INTERFACE I_MirrorCovers

METHOD Close : BOOL
VAR_INPUT
END_VAR
END_METHOD

PROPERTY Closed : BOOL
GET
END_GET
END_PROPERTY

PROPERTY Error : BOOL
GET
END_GET
END_PROPERTY

METHOD Open : BOOL
VAR_INPUT
END_VAR
END_METHOD

PROPERTY Opened : BOOL
GET
END_GET
END_PROPERTY

METHOD Reset : BOOL
VAR_INPUT
END_VAR
END_METHOD

END_INTERFACE

(* stored: Version 1.1.0.1, ProductVersion 3.1.4024.15
   Itf I_MirrorCovers: Id {ce637c3e-ed3e-4174-8b7f-5e29873c1a6c}
   Method Close: Id {154de5be-ed9e-40a6-affb-5973b8c678f6}
   Property Closed: Id {df5c5dcb-f0cb-4027-85a3-748560fa09dc}
   Get Get: Id {6a5afbac-a6cd-43df-90ce-766f647c9945}
   Property Error: Id {ff09ec7f-4b0d-4bfe-9bc0-a74f6b8e0c04}
   Get Get: Id {65d2e08e-b6f2-4c31-8697-8d42891b20d7}
   Method Open: Id {47330435-4ab9-4214-8907-9d0910956eeb}
   Property Opened: Id {9c791bb0-7b95-44f9-87e7-ce5d0e9a2540}
   Get Get: Id {fbdbf55f-40c4-4cdf-bbbf-a3b663be85c7}
   Method Reset: Id {8fd140fa-4504-401a-a6d2-edb6c92f8267} *)
